(* IEC 61131-3 sources: com.logicals.lc3.webinar/usRTS_RPMControl_iSOC/src_FB_LIB_SAFE/Timer, 3 files *)

(* ---- wTOF.iecst ---- *)
NAMESPACE logicals.web.standard
NAMESPACE timer

/*
 * Function block wrapper for IEC 61131-3 TOF<br>
 * IN = input, start (BOOL)<br>
 * PT = preset time (TIME)<br>
 * Q = output (BOOL)<br>
 * ET = elapsed time (TIME)<br>
 */
FUNCTION_BLOCK wTOF
	{ vNameAlignment:="center"; altName:="TOF"; bgColor:="YellowGreen"; width:=100; }
	VAR_INPUT
		IN : BOOL;
		PT : TIME;
	END_VAR
	VAR_OUTPUT
		Q  : BOOL;
		ET : TIME;
	END_VAR
	VAR
		TOF : TOF;
	END_VAR

	TOF(IN:=IN, PT:=PT, Q=>Q, ET=>ET, ENO=>ENO);
END_FUNCTION_BLOCK

END_NAMESPACE
END_NAMESPACE

(* ---- wTON.iecst ---- *)
NAMESPACE logicals.web.standard
NAMESPACE timer

/*
 * Function block wrapper for IEC 61131-3 TON<br>
 * IN = input, start (BOOL)<br>
 * PT = preset time (TIME)<br>
 * Q = output (BOOL)<br>
 * ET = elapsed time (TIME)<br>
 */
FUNCTION_BLOCK wTON
	{ vNameAlignment:="center"; altName:="TON"; bgColor:="YellowGreen"; width:=100; }
	VAR_INPUT
		IN : BOOL;
		PT : TIME;
	END_VAR
	VAR_OUTPUT
		Q  : BOOL;
		ET : TIME;
	END_VAR
	VAR
		TON : TON;
	END_VAR

	TON(IN:=IN, PT:=PT, Q=>Q, ET=>ET, ENO=>ENO);
END_FUNCTION_BLOCK

END_NAMESPACE
END_NAMESPACE

(* ---- wTP.iecst ---- *)
NAMESPACE logicals.web.standard
NAMESPACE timer

/*
 * Function block wrapper for IEC 61131-3 TP<br>
 * IN = input, start (BOOL)<br>
 * PT = preset time (TIME)<br>
 * Q = output (BOOL)<br>
 * ET = elapsed time (TIME)<br>
 */
FUNCTION_BLOCK wTP
	{ vNameAlignment:="center"; altName:="TP"; bgColor:="YellowGreen"; width:=100; }
	VAR_INPUT
		IN : BOOL;
		PT : TIME;
	END_VAR
	VAR_OUTPUT
		Q  : BOOL;
		ET : TIME;
	END_VAR
	VAR
		TP : TP;
	END_VAR

	TP(IN:=IN, PT:=PT, Q=>Q, ET=>ET, ENO=>ENO);
END_FUNCTION_BLOCK

END_NAMESPACE
END_NAMESPACE
